// TIA Portal V18 export
// export: Created 2026-06-24T03:56:38.0940771Z, ExportSetting WithDefaults, DisplayName Totally Integrated Automation Portal, DisplayVersion V18, DisplayName TIA Portal Openness, DisplayVersion V18, DisplayName TIA Portal Version Control Interface, DisplayVersion V18, DisplayName STEP 7 Professional, DisplayVersion V18, DisplayName STEP 7 Safety, DisplayVersion V18, DisplayName WinCC Professional, DisplayVersion V18
VAR_GLOBAL   // PLC tag table "Standard-Variablentabelle"
   start AT %I0.0 : Bool;
   stop AT %I0.1 : Bool;
   drain AT %I0.2 : Bool;
   levelMeter AT %ID30 : Real;
   SetPoint AT %ID38 : Real;
   FillValve AT %QD30 : Real;
   DissValve AT %QD34 : Real;
   SetPointDisplay AT %QD38 : DInt;
   LevelDisplay AT %QD42 : DInt;
   ErrorDisplay AT %QD46 : Real;
   Tag_1 AT %M0.0 : Bool;
   Tag_2 AT %MD100 : Real;
   scaledlevel AT %MW2 : Int;
   setscaled AT %MW12 : Int;
   Tag_3 AT %M2.2 : Bool;
END_VAR
